{attribute addProperty BoxType "EP7041-0002-0016"}
{attribute addProperty Id "ControlAT %Q*Control_D763B95710012.5"}
{attribute addProperty CRC "3420697581"}
{attribute addProperty SizeInBites "100"}
{attribute addProperty SizeInBytes "12.5"}
TYPE STM_Control_CBE3B3ED :
STRUCT
	{attribute addProperty Name "Control"}
	Control AT %Q* : Control_D763B957;
END_STRUCT
END_TYPE

(* stored: Version 1.2.0.0, ProductVersion 3.1.4024.9
   DUT STM_Control_CBE3B3ED: Id {ea87d3fa-360f-4d1d-8ee6-cd5296e025f5} *)
